FUNCTION CELSIUS_TO_KELVIN : REAL
VAR_INPUT
    celsius : REAL;
END_VAR
VAR
END_VAR

CELSIUS_TO_KELVIN := celsius + 273.15;

END_FUNCTION

(* stored: Version 1.1.0.1, ProductVersion 3.1.4018.5
   POU CELSIUS_TO_KELVIN: Id {d26afcbc-1881-4acd-898c-728619f3a1f3}, SpecialFunc None *)
